VISUALIZATION LED_visu  // 2x2
VAR_IN_OUT
	bLED1	: BOOL;
END_VAR
END_VISUALIZATION

(* stored: Version 1.1.0.1, ProductVersion 3.1.4022.3
   Visu LED_visu: Id {ac26332f-a287-48e4-8993-3ef20bde8bd4} *)
